TYPE
    WcState :
    STRUCT
        WcState : BIT; // 0 valid
        InputToggle   : BIT;
    END_STRUCT
END_TYPE

(* stored: Version 1.1.0.1, ProductVersion 3.1.4024.12
   DUT WcState: Id {e7b95519-5761-4d8f-9803-0f2a8adca8b7} *)
